// TIA Portal V20 export
TYPE "typeSafetyZoneStatus"
// Status of safety zone
// stored: Access Published, IsFailsafeCompliant true, Namespace Safety
   STRUCT
      safetyReleased1 { ExternalWritable := 'False'} : Bool;   // Safety zone is released_SS1
      safetyReleased2 { ExternalWritable := 'False'} : Bool;   // Safety zone is released_SS2
      ackReq { ExternalWritable := 'False'} : Bool;   // Acknowledge is required
      safetyFault { ExternalWritable := 'False'} : Bool;   // Safety fault in at least one device is active
      highSpeedEnable { ExternalWritable := 'False'} : Bool;   // SLS : Normal On
      activeSLS { ExternalWritable := 'False'} : Bool;   // SLS is activated on Zone
      activeSTO { ExternalWritable := 'False'} : Bool;   // STO is activated on Zone
      activeSOS { ExternalWritable := 'False'} : Bool;   // STO is activated on Zone
      activeSS1 { ExternalWritable := 'False'} : Bool;   // STO is activated on Zone
      activeSS2 { ExternalWritable := 'False'} : Bool;   // STO is activated on Zone
      AllFDoorClose : Bool;   // All Door Close
      SFDoorOpen { ExternalWritable := 'False'} : Bool;   // Only One Door Open
      MFDoorOpen { ExternalWritable := 'False'} : Bool;   // Multi Door Open
   END_STRUCT;
END_TYPE
